(* PLC project  *)

CONFIGURATION Empty_Module_16
END_CONFIGURATION
